PROGRAM stMain	
VAR

	OUT_VAL:	REAL := 0;	
	
	T1:	TON;
END_VAR


T1(IN:=(T1.Q=FALSE),PT:=T#1.0S,);

IF T1.Q THEN

	AOUT[1]		:= REAL_TO_INT(OUT_VAL);
	AOUT[2]		:= REAL_TO_INT(4*OUT_VAL);
	
	OUT_VAL := OUT_VAL + 100.0;
	
	IF (OUT_VAL > 32768.0/8.0) THEN
		OUT_VAL := 0;
	END_IF
	
END_IF

END_PROGRAM

(* stored: Version 1.1.0.1, ProductVersion 3.1.0.36
   POU stMain: Id {209e7332-f57a-4ce8-887e-f94efce2de36}, SpecialFunc None *)
